FUNCTION F_AlarmPrioToHexColor : STRING
VAR_INPUT
	ePriority : E_AlarmPriority;
END_VAR

			
CASE ePriority OF
	E_AlarmPriority.Error:
		F_AlarmPrioToHexColor := F_ColorToStringHexColor(STATICS.stColor.Red);
		
	E_AlarmPriority.Warning:
		F_AlarmPrioToHexColor := F_ColorToStringHexColor(STATICS.stColor.Orange);
		
	ELSE
		F_AlarmPrioToHexColor := F_ColorToStringHexColor(STATICS.stColor.Blue); //F_ColorToStringHexColor(stCol.Theme);
	
END_CASE

END_FUNCTION

(* stored: Version 1.1.0.1, ProductVersion 3.1.4024.12
   POU F_AlarmPrioToHexColor: Id {8cf0b548-190c-42c6-8820-067a3def7903}, SpecialFunc None *)
